END_VAR
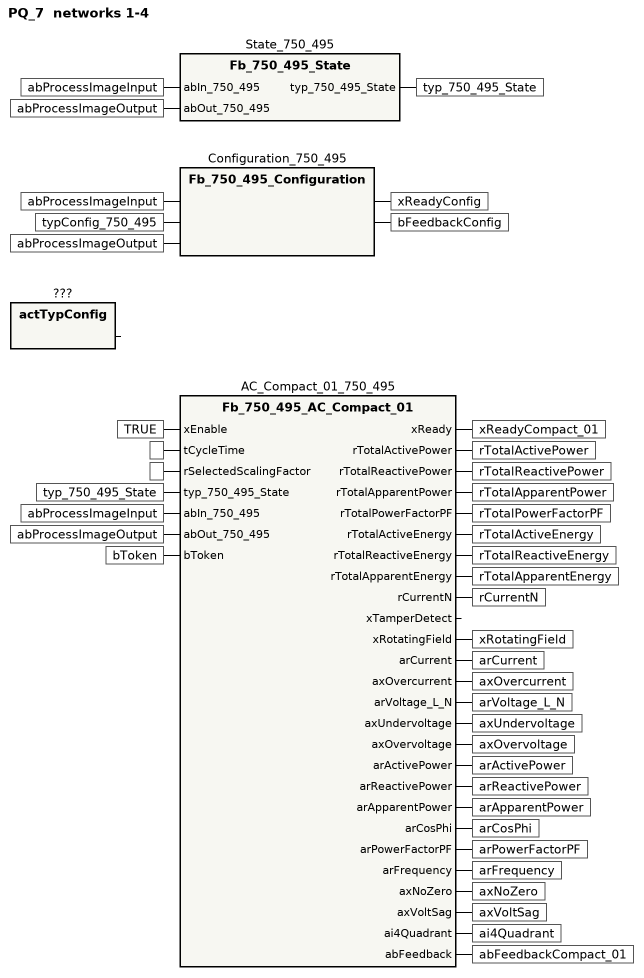
[picture p21: PQ_7 (FBD) networks 1-4]
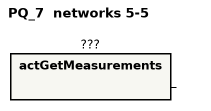
_FBD_ (* Function Block Diagram *)
NETWORK 1
	State_750_495:Fb_750_495_State(abIn_750_495: abProcessImageInput, abOut_750_495: abProcessImageOutput) => typ_750_495_State
NETWORK 2
	Configuration_750_495:Fb_750_495_Configuration(abProcessImageInput, typConfig_750_495, abProcessImageOutput, out 2 => bFeedbackConfig) => xReadyConfig
NETWORK 3
	???:actTypConfig()
NETWORK 4
	AC_Compact_01_750_495:Fb_750_495_AC_Compact_01(xEnable: TRUE, tCycleTime: , rSelectedScalingFactor: , typ_750_495_State: typ_750_495_State, abIn_750_495: abProcessImageInput, abOut_750_495: abProcessImageOutput, bToken: bToken, rTotalActivePower => rTotalActivePower, rTotalReactivePower => rTotalReactivePower, rTotalApparentPower => rTotalApparentPower, rTotalPowerFactorPF => rTotalPowerFactorPF, rTotalActiveEnergy => rTotalActiveEnergy, rTotalReactiveEnergy => rTotalReactiveEnergy, rTotalApparentEnergy => rTotalApparentEnergy, rCurrentN => rCurrentN, xRotatingField => xRotatingField, arCurrent => arCurrent, axOvercurrent => axOvercurrent, arVoltage_L_N => arVoltage_L_N, axUndervoltage => axUndervoltage, axOvervoltage => axOvervoltage, arActivePower => arActivePower, arReactivePower => arReactivePower, arApparentPower => arApparentPower, arCosPhi => arCosPhi, arPowerFactorPF => arPowerFactorPF, arFrequency => arFrequency, axNoZero => axNoZero, axVoltSag => axVoltSag, ai4Quadrant => ai4Quadrant, abFeedback => abFeedbackCompact_01) => xReadyCompact_01
NETWORK 5
	???:actGetMeasurements()
_END_FBD_
(* the same logic as Structured Text *)
(* Network 1 *)
State_750_495(abIn_750_495 := abProcessImageInput, abOut_750_495 := abProcessImageOutput);
typ_750_495_State := State_750_495.typ_750_495_State;
(* Network 2: see the listing above *)
(* Network 3: see the listing above *)
(* Network 4: see the listing above *)
(* Network 5: see the listing above *)
END_PROGRAM
ACTION actGetMeasurements:
arMeasurementsGroup7[1] := arActivePower[1];
arMeasurementsGroup7[2] := arActivePower[2];
arMeasurementsGroup7[3] := arActivePower[3];
arMeasurementsGroup7[4] := arReactivePower[1];
arMeasurementsGroup7[5] := arReactivePower[2];
arMeasurementsGroup7[6] := arReactivePower[3];
arMeasurementsGroup7[7] := arVoltage_L_N[1];
arMeasurementsGroup7[8] := arVoltage_L_N[2];
arMeasurementsGroup7[9] := arVoltage_L_N[3];
arMeasurementsGroup7[10] := arCurrent[1];
arMeasurementsGroup7[11] := arCurrent[2];
arMeasurementsGroup7[12] := arCurrent[3];
arMeasurementsGroup7[13] := arFrequency[1];
arMeasurementsGroup7[14] := arFrequency[2];
arMeasurementsGroup7[15] := arFrequency[3];
arMeasurementsGroup7[16] := rTotalActiveEnergy;
arMeasurementsGroup7[17] := BOOL_TO_REAL(xRotatingField);
arMeasurementsGroup7[18] := rTotalReactiveEnergy;
END_ACTION
ACTION actTypConfig:
typConfig_750_495.typChannelConfig[1].xEnableUserScaling:= TRUE;
typConfig_750_495.typChannelConfig[1].wCurrentTransformerRatio :=CurrentRatioPQ1;

typConfig_750_495.typChannelConfig[2].xEnableUserScaling:= TRUE;
typConfig_750_495.typChannelConfig[2].wCurrentTransformerRatio :=CurrentRatioPQ1;

typConfig_750_495.typChannelConfig[3].xEnableUserScaling:= TRUE;
typConfig_750_495.typChannelConfig[3].wCurrentTransformerRatio :=CurrentRatioPQ1;

typConfig_750_495.xWriteConfig := TRUE;
END_ACTION

(* POU 01. PowerQualityMeasurements/PQ_8, FBD *)
PROGRAM PQ_8
VAR
	abProcessImageInput	AT %IW96			: ARRAY[0..23] OF BYTE;
	abProcessImageOutput 	AT %QW104 		: ARRAY[0..23] OF BYTE;

	bToken										: BYTE;

	State_750_495 							: Fb_750_495_State;
		typ_750_495_State 						: typ_750_495_State;

	Configuration_750_495					: Fb_750_495_Configuration;
		typConfig_750_495						: typConfig_750_495;
		xReadyConfig								: BOOL;
		bFeedbackConfig							: BYTE;

	AC_Compact_01_750_495				: Fb_750_495_AC_Compact_01;
		rTotalActivePower							: REAL;
		rTotalReactivePower						: REAL;
		rTotalApparentPower						: REAL;
		rTotalPowerFactorPF						: REAL;
		rTotalActiveEnergy							: REAL;
		rTotalReactiveEnergy						: REAL;
		rTotalApparentEnergy						: REAL;
		rCurrentN									: REAL;
		xRotatingField								: BOOL;
		arCurrent									: ARRAY[1..3] OF REAL;
		axOvercurrent								: ARRAY[1..3] OF BOOL;
		arVoltage_L_N							: ARRAY[1..3] OF REAL;
		axUndervoltage							: ARRAY[1..3] OF BOOL;
		axOvervoltage								: ARRAY[1..3] OF BOOL;
		arActivePower								: ARRAY[1..3] OF REAL;
		arReactivePower							: ARRAY[1..3] OF REAL;
		arApparentPower							: ARRAY[1..3] OF REAL;
		arCosPhi									: ARRAY[1..3] OF REAL;
		arPowerFactorPF							: ARRAY[1..3] OF REAL;
		arFrequency								: ARRAY[1..3] OF REAL;
		axNoZero									: ARRAY[1..3] OF BOOL;
		axVoltSag									: ARRAY[1..3] OF BOOL;
		ai4Quadrant								: ARRAY[1..3] OF INT;

		xReadyCompact_01						: BOOL;
		abFeedbackCompact_01					: ARRAY[1..8] OF BYTE;


END_VAR
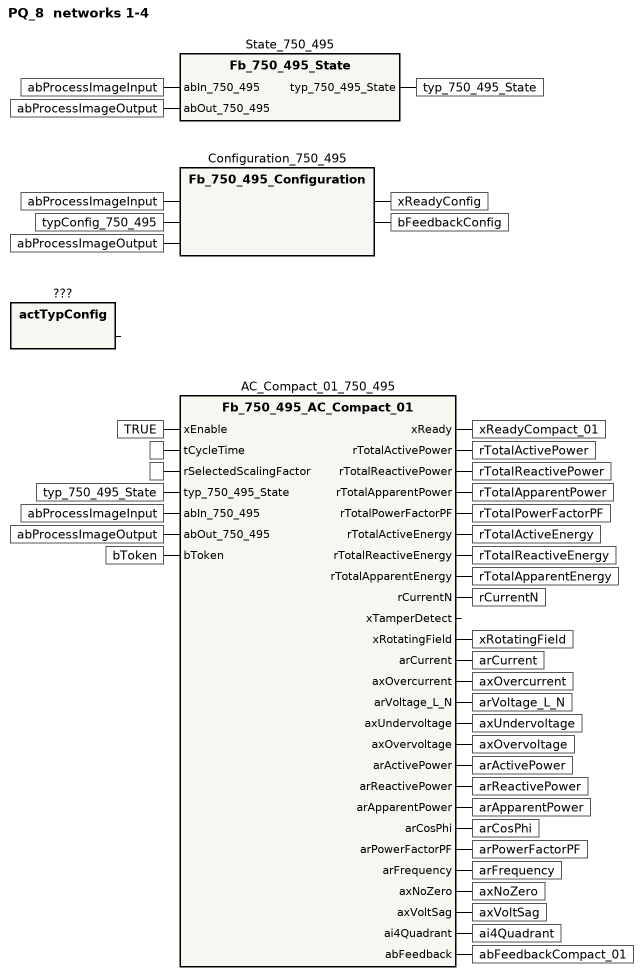
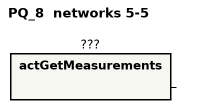
_FBD_ (* Function Block Diagram *)
NETWORK 1
	State_750_495:Fb_750_495_State(abIn_750_495: abProcessImageInput, abOut_750_495: abProcessImageOutput) => typ_750_495_State
NETWORK 2
	Configuration_750_495:Fb_750_495_Configuration(abProcessImageInput, typConfig_750_495, abProcessImageOutput, out 2 => bFeedbackConfig) => xReadyConfig
NETWORK 3
	???:actTypConfig()
NETWORK 4
	AC_Compact_01_750_495:Fb_750_495_AC_Compact_01(xEnable: TRUE, tCycleTime: , rSelectedScalingFactor: , typ_750_495_State: typ_750_495_State, abIn_750_495: abProcessImageInput, abOut_750_495: abProcessImageOutput, bToken: bToken, rTotalActivePower => rTotalActivePower, rTotalReactivePower => rTotalReactivePower, rTotalApparentPower => rTotalApparentPower, rTotalPowerFactorPF => rTotalPowerFactorPF, rTotalActiveEnergy => rTotalActiveEnergy, rTotalReactiveEnergy => rTotalReactiveEnergy, rTotalApparentEnergy => rTotalApparentEnergy, rCurrentN => rCurrentN, xRotatingField => xRotatingField, arCurrent => arCurrent, axOvercurrent => axOvercurrent, arVoltage_L_N => arVoltage_L_N, axUndervoltage => axUndervoltage, axOvervoltage => axOvervoltage, arActivePower => arActivePower, arReactivePower => arReactivePower, arApparentPower => arApparentPower, arCosPhi => arCosPhi, arPowerFactorPF => arPowerFactorPF, arFrequency => arFrequency, axNoZero => axNoZero, axVoltSag => axVoltSag, ai4Quadrant => ai4Quadrant, abFeedback => abFeedbackCompact_01) => xReadyCompact_01
NETWORK 5
	???:actGetMeasurements()
_END_FBD_
(* the same logic as Structured Text *)
(* Network 1 *)
State_750_495(abIn_750_495 := abProcessImageInput, abOut_750_495 := abProcessImageOutput);
typ_750_495_State := State_750_495.typ_750_495_State;
(* Network 2: see the listing above *)
(* Network 3: see the listing above *)
(* Network 4: see the listing above *)
(* Network 5: see the listing above *)
END_PROGRAM
ACTION actGetMeasurements:
arMeasurementsGroup8[1] := arActivePower[1];
arMeasurementsGroup8[2] := arActivePower[2];
arMeasurementsGroup8[3] := arActivePower[3];
arMeasurementsGroup8[4] := arReactivePower[1];
arMeasurementsGroup8[5] := arReactivePower[2];
arMeasurementsGroup8[6] := arReactivePower[3];
arMeasurementsGroup8[7] := arVoltage_L_N[1];
arMeasurementsGroup8[8] := arVoltage_L_N[2];
arMeasurementsGroup8[9] := arVoltage_L_N[3];
arMeasurementsGroup8[10] := arCurrent[1];
arMeasurementsGroup8[11] := arCurrent[2];
arMeasurementsGroup8[12] := arCurrent[3];
arMeasurementsGroup8[13] := arFrequency[1];
arMeasurementsGroup8[14] := arFrequency[2];
arMeasurementsGroup8[15] := arFrequency[3];
arMeasurementsGroup8[16] := rTotalActiveEnergy;
arMeasurementsGroup8[17] := BOOL_TO_REAL(xRotatingField);
arMeasurementsGroup8[18] := rTotalReactiveEnergy;
END_ACTION
ACTION actTypConfig:
typConfig_750_495.typChannelConfig[1].xEnableUserScaling:= TRUE;
typConfig_750_495.typChannelConfig[1].wCurrentTransformerRatio :=CurrentRatioPQ1;

typConfig_750_495.typChannelConfig[2].xEnableUserScaling:= TRUE;
typConfig_750_495.typChannelConfig[2].wCurrentTransformerRatio :=CurrentRatioPQ1;

typConfig_750_495.typChannelConfig[3].xEnableUserScaling:= TRUE;
typConfig_750_495.typChannelConfig[3].wCurrentTransformerRatio :=CurrentRatioPQ1;

typConfig_750_495.xWriteConfig := TRUE;
END_ACTION

(* POU 01. PowerQualityMeasurements/PQ_9, FBD *)
PROGRAM PQ_9
VAR
	abProcessImageInput	AT %IW108		: ARRAY[0..23] OF BYTE;
	abProcessImageOutput 	AT %QW116		: ARRAY[0..23] OF BYTE;

	bToken										: BYTE;

	State_750_495 							: Fb_750_495_State;
		typ_750_495_State 						: typ_750_495_State;

	Configuration_750_495					: Fb_750_495_Configuration;
		typConfig_750_495						: typConfig_750_495;
		xReadyConfig								: BOOL;
		bFeedbackConfig							: BYTE;

	AC_Compact_01_750_495				: Fb_750_495_AC_Compact_01;
		rTotalActivePower							: REAL;
		rTotalReactivePower						: REAL;
		rTotalApparentPower						: REAL;
		rTotalPowerFactorPF						: REAL;
		rTotalActiveEnergy							: REAL;
		rTotalReactiveEnergy						: REAL;
		rTotalApparentEnergy						: REAL;
		rCurrentN									: REAL;
		xRotatingField								: BOOL;
		arCurrent									: ARRAY[1..3] OF REAL;
		axOvercurrent								: ARRAY[1..3] OF BOOL;
		arVoltage_L_N							: ARRAY[1..3] OF REAL;
		axUndervoltage							: ARRAY[1..3] OF BOOL;
		axOvervoltage								: ARRAY[1..3] OF BOOL;
		arActivePower								: ARRAY[1..3] OF REAL;
		arReactivePower							: ARRAY[1..3] OF REAL;
		arApparentPower							: ARRAY[1..3] OF REAL;
		arCosPhi									: ARRAY[1..3] OF REAL;
		arPowerFactorPF							: ARRAY[1..3] OF REAL;
		arFrequency								: ARRAY[1..3] OF REAL;
		axNoZero									: ARRAY[1..3] OF BOOL;
		axVoltSag									: ARRAY[1..3] OF BOOL;
		ai4Quadrant								: ARRAY[1..3] OF INT;

		xReadyCompact_01						: BOOL;
		abFeedbackCompact_01					: ARRAY[1..8] OF BYTE;


END_VAR
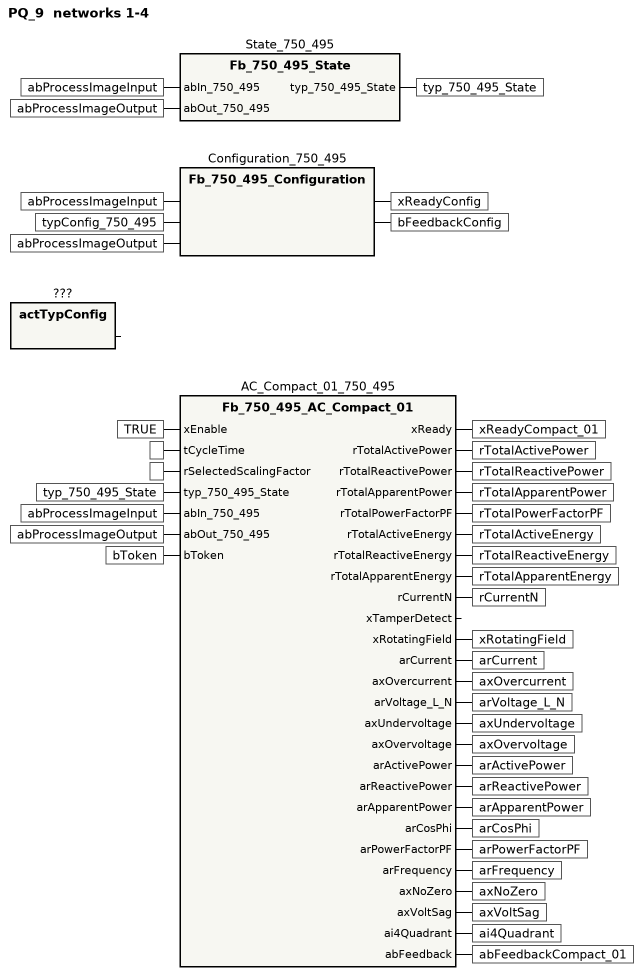
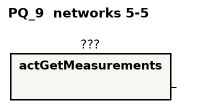
_FBD_ (* Function Block Diagram *)
NETWORK 1
	State_750_495:Fb_750_495_State(abIn_750_495: abProcessImageInput, abOut_750_495: abProcessImageOutput) => typ_750_495_State
NETWORK 2
	Configuration_750_495:Fb_750_495_Configuration(abProcessImageInput, typConfig_750_495, abProcessImageOutput, out 2 => bFeedbackConfig) => xReadyConfig
NETWORK 3
	???:actTypConfig()
NETWORK 4
	AC_Compact_01_750_495:Fb_750_495_AC_Compact_01(xEnable: TRUE, tCycleTime: , rSelectedScalingFactor: , typ_750_495_State: typ_750_495_State, abIn_750_495: abProcessImageInput, abOut_750_495: abProcessImageOutput, bToken: bToken, rTotalActivePower => rTotalActivePower, rTotalReactivePower => rTotalReactivePower, rTotalApparentPower => rTotalApparentPower, rTotalPowerFactorPF => rTotalPowerFactorPF, rTotalActiveEnergy => rTotalActiveEnergy, rTotalReactiveEnergy => rTotalReactiveEnergy, rTotalApparentEnergy => rTotalApparentEnergy, rCurrentN => rCurrentN, xRotatingField => xRotatingField, arCurrent => arCurrent, axOvercurrent => axOvercurrent, arVoltage_L_N => arVoltage_L_N, axUndervoltage => axUndervoltage, axOvervoltage => axOvervoltage, arActivePower => arActivePower, arReactivePower => arReactivePower, arApparentPower => arApparentPower, arCosPhi => arCosPhi, arPowerFactorPF => arPowerFactorPF, arFrequency => arFrequency, axNoZero => axNoZero, axVoltSag => axVoltSag, ai4Quadrant => ai4Quadrant, abFeedback => abFeedbackCompact_01) => xReadyCompact_01
NETWORK 5
	???:actGetMeasurements()
_END_FBD_
(* the same logic as Structured Text *)
(* Network 1 *)
State_750_495(abIn_750_495 := abProcessImageInput, abOut_750_495 := abProcessImageOutput);
typ_750_495_State := State_750_495.typ_750_495_State;
(* Network 2: see the listing above *)
(* Network 3: see the listing above *)
(* Network 4: see the listing above *)
(* Network 5: see the listing above *)
END_PROGRAM
ACTION actGetMeasurements:
arMeasurementsGroup9[1] := arActivePower[1];
arMeasurementsGroup9[2] := arActivePower[2];
arMeasurementsGroup9[3] := arActivePower[3];
arMeasurementsGroup9[4] := arReactivePower[1];
arMeasurementsGroup9[5] := arReactivePower[2];
arMeasurementsGroup9[6] := arReactivePower[3];
arMeasurementsGroup9[7] := arVoltage_L_N[1];
arMeasurementsGroup9[8] := arVoltage_L_N[2];
arMeasurementsGroup9[9] := arVoltage_L_N[3];
arMeasurementsGroup9[10] := arCurrent[1];
arMeasurementsGroup9[11] := arCurrent[2];
arMeasurementsGroup9[12] := arCurrent[3];
arMeasurementsGroup9[13] := arFrequency[1];
arMeasurementsGroup9[14] := arFrequency[2];
arMeasurementsGroup9[15] := arFrequency[3];
arMeasurementsGroup9[16] := rTotalActiveEnergy;
arMeasurementsGroup9[17] := BOOL_TO_REAL(xRotatingField);
arMeasurementsGroup9[18] := rTotalReactiveEnergy;
END_ACTION
ACTION actTypConfig:
typConfig_750_495.typChannelConfig[1].xEnableUserScaling:= TRUE;
typConfig_750_495.typChannelConfig[1].wCurrentTransformerRatio :=CurrentRatioPQ1;

typConfig_750_495.typChannelConfig[2].xEnableUserScaling:= TRUE;
typConfig_750_495.typChannelConfig[2].wCurrentTransformerRatio :=CurrentRatioPQ1;

typConfig_750_495.typChannelConfig[3].xEnableUserScaling:= TRUE;
typConfig_750_495.typChannelConfig[3].wCurrentTransformerRatio :=CurrentRatioPQ1;

typConfig_750_495.xWriteConfig := TRUE;
END_ACTION

(* POU 02. Batterybus Frequency to Analog Out/CHP_Controller, FBD *)
PROGRAM CHP_Controller
VAR
	RAMP_REAL: RAMP_REAL;
	Frequency_to_Analog_Out: Frequency_to_Analog_Out;
END_VAR
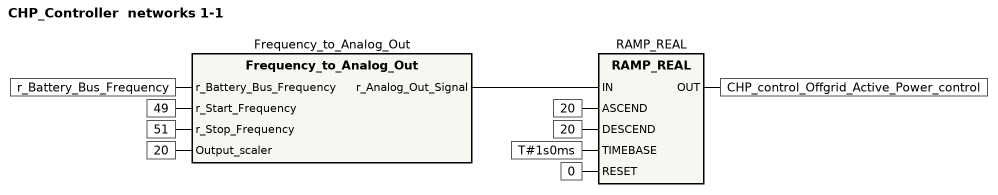
_FBD_ (* Function Block Diagram *)
NETWORK 1
	RAMP_REAL:RAMP_REAL(IN: Frequency_to_Analog_Out:Frequency_to_Analog_Out(r_Battery_Bus_Frequency: r_Battery_Bus_Frequency, r_Start_Frequency: 49, r_Stop_Frequency: 51, Output_scaler: 20), ASCEND: 20, DESCEND: 20, TIMEBASE: T#1s0ms, RESET: 0) => CHP_control_Offgrid_Active_Power_control
_END_FBD_
(* the same logic as Structured Text *)
(* Network 1 *)
Frequency_to_Analog_Out(r_Battery_Bus_Frequency := r_Battery_Bus_Frequency, r_Start_Frequency := 49, r_Stop_Frequency := 51, Output_scaler := 20);
RAMP_REAL(IN := Frequency_to_Analog_Out.r_Analog_Out_Signal, ASCEND := 20, DESCEND := 20, TIMEBASE := T#1s0ms, RESET := 0);
CHP_control_Offgrid_Active_Power_control := RAMP_REAL.OUT;
END_PROGRAM

(* POU 02. Batterybus Frequency to Analog Out/Frequency_to_Analog_Out, ST *)
FUNCTION_BLOCK Frequency_to_Analog_Out
VAR_INPUT
	r_Battery_Bus_Frequency						:	REAL;
	r_Start_Frequency								:	REAL:=49;
	r_Stop_Frequency								:	REAL:=51;
	Output_scaler										:	REAL:=1;
END_VAR

VAR_OUTPUT
	r_Analog_Out_Signal								:	REAL;
END_VAR

VAR

END_VAR
(* limit control range inbetween start/stop input*)
IF r_Start_Frequency < r_Stop_Frequency THEN
	IF r_Battery_Bus_Frequency < r_Start_Frequency THEN
			r_Battery_Bus_Frequency := r_Start_Frequency;
	END_IF
	IF r_Battery_Bus_Frequency > r_Stop_Frequency THEN
			r_Battery_Bus_Frequency := r_Stop_Frequency;
	END_IF
ELSE
	IF r_Battery_Bus_Frequency > r_Start_Frequency THEN
			r_Battery_Bus_Frequency := r_Start_Frequency;
	END_IF
	IF r_Battery_Bus_Frequency < r_Stop_Frequency THEN
			r_Battery_Bus_Frequency := r_Stop_Frequency;
	END_IF
END_IF

r_Analog_Out_Signal := (r_Battery_Bus_Frequency - r_Start_Frequency) / (r_Stop_Frequency - r_Start_Frequency) * Output_scaler;
END_FUNCTION_BLOCK

(* POU 02. Batterybus Frequency to Analog Out/EV_Controller, FBD *)
PROGRAM EV_Controller
VAR
	RAMP_REAL: RAMP_REAL;
	Frequency_to_Analog_Out: Frequency_to_Analog_Out;
END_VAR
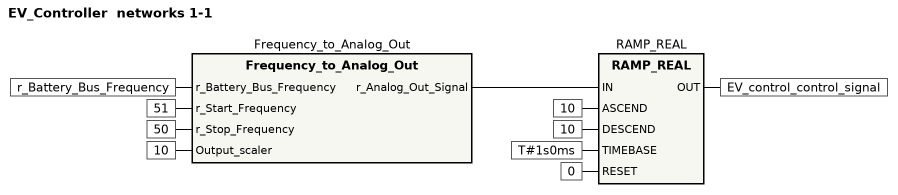
_FBD_ (* Function Block Diagram *)
NETWORK 1
	RAMP_REAL:RAMP_REAL(IN: Frequency_to_Analog_Out:Frequency_to_Analog_Out(r_Battery_Bus_Frequency: r_Battery_Bus_Frequency, r_Start_Frequency: 51, r_Stop_Frequency: 50, Output_scaler: 10), ASCEND: 10, DESCEND: 10, TIMEBASE: T#1s0ms, RESET: 0) => EV_control_control_signal
_END_FBD_
(* the same logic as Structured Text *)
(* Network 1 *)
Frequency_to_Analog_Out(r_Battery_Bus_Frequency := r_Battery_Bus_Frequency, r_Start_Frequency := 51, r_Stop_Frequency := 50, Output_scaler := 10);
RAMP_REAL(IN := Frequency_to_Analog_Out.r_Analog_Out_Signal, ASCEND := 10, DESCEND := 10, TIMEBASE := T#1s0ms, RESET := 0);
EV_control_control_signal := RAMP_REAL.OUT;
END_PROGRAM

(* POU 02. Batterybus Frequency to Analog Out/Mixer_Controller, FBD *)
PROGRAM Mixer_Controller
VAR
	RAMP_REAL: RAMP_REAL;
	Frequency_to_Analog_Out: Frequency_to_Analog_Out;
END_VAR
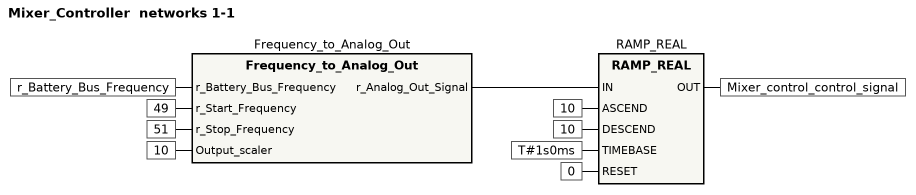
_FBD_ (* Function Block Diagram *)
NETWORK 1
	RAMP_REAL:RAMP_REAL(IN: Frequency_to_Analog_Out:Frequency_to_Analog_Out(r_Battery_Bus_Frequency: r_Battery_Bus_Frequency, r_Start_Frequency: 49, r_Stop_Frequency: 51, Output_scaler: 10), ASCEND: 10, DESCEND: 10, TIMEBASE: T#1s0ms, RESET: 0) => Mixer_control_control_signal
_END_FBD_
(* the same logic as Structured Text *)
(* Network 1 *)
Frequency_to_Analog_Out(r_Battery_Bus_Frequency := r_Battery_Bus_Frequency, r_Start_Frequency := 49, r_Stop_Frequency := 51, Output_scaler := 10);
RAMP_REAL(IN := Frequency_to_Analog_Out.r_Analog_Out_Signal, ASCEND := 10, DESCEND := 10, TIMEBASE := T#1s0ms, RESET := 0);
Mixer_control_control_signal := RAMP_REAL.OUT;
END_PROGRAM

(* POU PLC_PRG, FBD *)
PROGRAM PLC_PRG
(*
  Function: 	Reading a CSV file
  Description: 	This project shows a functionblock which reads data from a CSV file into an array.
				Each line in the CSV contains a description and a real value.
				Each parameter  is terminated by CR LF.

---- Example CSV File -----

A_Value;245345
B_Value;0							
C_Value;8.3							
D_Value;-123439.3 						
E_Value;1						*)

VAR
	xLoad					: 	BOOL; (* Initiate load operation *)
	xSave					: 	BOOL; (* Initiate save operation *)
	sLoadStatus			: 	STRING; (* Feedback on load *)
	sSaveStatus			: 	STRING; (* Feedback on save *)
	ConfigData			: 	ARRAY [1..iMaxParams] OF  typCSV; (* Structure with the config data being loaded or saved *)
	sFileName			: 	STRING := 'config.csv'; (* Working Filename *)
	bSeperator 			: 	BYTE := 59; (* Semicolon (;) is the seperator between parameter and value. *)
	iError					: 	INT; (* Error Code for Save *)
	xWriteToSD			: 	BOOL := TRUE; (* User selectable location for file operation, on = 750-880 SD, off = internal flash *)
	sFilePath				: 	STRING; (* SD card is S:\, Internal Path is blank, but this points to the PLC folder *)
	sFilePath_Name		: 	STRING; (* Complete path + filename *)

	xReadFirstCycle		:	BOOL := TRUE;

	SetIPConfig				:	configToolFB;
	SetIP						:	configToolFB;
	SetSubnet					:	configToolFB;
	SetGateway				:	configToolFB;
	SetNTP					:	configToolFB;
	SetNTPEnable			:	configToolFB;
	SetSNMPName			:	configToolFB;
	SetSNMPDescription		:	configToolFB;
	SetSNMPLocation			:	configToolFB;
	SetSNMPContact			:	configToolFB;

	GetIPConfig				:	configToolFB;
	GetIP						:	configToolFB;
	GetSubnet					:	configToolFB;
	GetGateway				:	configToolFB;
	GetNTP					:	configToolFB;
	GetSNMPName			:	configToolFB;
	GetSNMPDescription		:	configToolFB;
	GetSNMPLocation		:	configToolFB;
	GetSNMPContact			:	configToolFB;
	GetFirmware				:	configToolFB;
	GetMACAddress			:	configToolFB;
	GetProjectDate			:	configToolFB;
	GetProjectDescription	:	configToolFB;
	GetProjectVersion			:	configToolFB;

	stSetIPConfigCallstring				:	STRING(80);
	stSetIPCallstring						:	STRING(80);
	stSetSubnetCallstring				:	STRING(80);
	stSetGatewayCallstring				:	STRING(80);
	stSetNTPCallstring					:	STRING(80);

	iSetIPConfigCallstringResult			:	INT;
	iSetIPCallstringResult				:	INT;
	iSetSubnetCallstringResult			:	INT;
	iSetGatewayCallstringResult			:	INT;
	iSetNTPCallstringResult				: 	INT;
	iSetNTPEnabledCallstringResult	:	INT;

	iGetIPConfigCallstringResult			:	INT;
	iGetIPCallstringResult				:	INT;
	iGetSubnetCallstringResult			:	INT;
	iGetGatewayCallstringResult			:	INT;
	iGetNTPCallstringResult				: 	INT;
	iGetNTPEnabledCallstringResult	:	INT;

	iGetFirmwareCallstringResult				:	INT;
	iGetMACAddressCallstringResult			:	INT;
	iGetProjectDateCallstringResult				:	INT;
	iGetProjectDescriptionCallstringResult		:	INT;
	iGetProjectVersionCallstringResult			:	INT;

	stGetIPConfigCallstring				:	STRING(80);
	stGetIPCallstring						:	STRING(80);
	stGetSubnetCallstring				:	STRING(80);
	stGetGatewayCallstring				:	STRING(80);
	stGetNTPCallstring					:	STRING(80);

	stSetIPConfigResult					:	STRING(80);
	stSetIPResult							:	STRING(80);
	stSetSubnetResult					:	STRING(80);
	stSetGatewayResult					:	STRING(80);
	stSetNTPResult						:	STRING(80);

	stGetIPConfigResult					:	STRING(80);
	stGetIPResult							:	STRING(80);
	stGetSubnetResult					:	STRING(80);
	stGetGatewayResult					:	STRING(80);
	stGetNTPResult						:	STRING(80);

	stSetSNMPNameDeviceCallstring					:	STRING(80);
	stSetSNMPDescriptionCallstring						:	STRING(80);
	stSetSNMPPhysicalLocationCallstring				:	STRING(80);
	stSetSNMPContactCallstring							:	STRING(80);

	stGetSNMPNameDeviceResult						:	STRING(80);
	stGetSNMPDescriptionResult						:	STRING(80);
	stGetSNMPPhysicalLocationResult					:	STRING(80);
	stGetSNMPContactResult							:	STRING(80);

	stGetFirmwareResult									:	STRING(80);
	stGetMACAddressResult								:	STRING(80);
	stGetProjectDateResult								:	STRING(80);
	stGetProjectDescriptionResult						:	STRING(80);
	stGetProjectVersionResult							:	STRING(80);

	iSetSNMPNameDeviceCallstringResult				:	INT;
	iSetSNMPDescriptionCallstringResult				:	INT;
	iSetSNMPPhysicalLocationCallstringResult			:	INT;
	iSetSNMPContactCallstringResult					:	INT;

	iGetSNMPNameDeviceCallstringResult				:	INT;
	iGetSNMPDescriptionCallstringResult				:	INT;
	iGetSNMPPhysicalLocationCallstringResult			:	INT;
	iGetSNMPContactCallstringResult					:	INT;

	CurrentTimeDate										:	STRING;

END_VAR
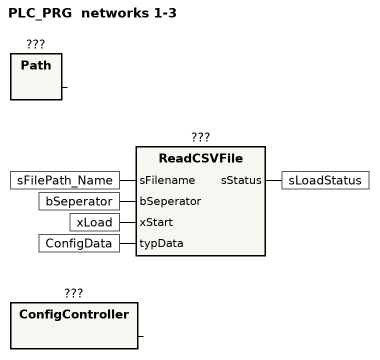
_FBD_ (* Function Block Diagram *)
NETWORK 1
	???:Path()
NETWORK 2
	???:ReadCSVFile(sFilename: sFilePath_Name, bSeperator: bSeperator, xStart: xLoad, typData: ConfigData) => sLoadStatus
NETWORK 3
	???:ConfigController()
_END_FBD_
END_PROGRAM
ACTION ConfigController:
IF xReadFirstCycle = TRUE THEN

	(*xLoad := TRUE;*)

	IF sLoadStatus = 'Data read OK' THEN
	
		(* Set Ethernet settings of controller *)
		
		(* Set static IP-Address*)
		
		
			SetIPConfig(
			bEnable:= TRUE,
			stCallString:= 'config_interfaces interface=X1 config-type=static state=enabled',
			stResultString=> stSetIPConfigResult,
			iFbResult=> iSetIPCallstringResult );
		
		(* Set IP-Address of controller *)
		
			stSetIPCallstring := CONCAT('config_interfaces interface X1 ip-address=',stIPAddressEthernet);
		
			SetIP(
			bEnable:= TRUE,
			stCallString:= stSetIPCallstring ,
			stResultString=> stSetIPResult,
			iFbResult=> iSetIPCallstringResult );
		
		(* Set Subnet-Address of controller *)
		
			stSetSubnetCallstring := CONCAT('config_interfaces interface X1 subnet-mask=',stIPAddressSubnet);
		
			SetSubnet(
			bEnable:= TRUE,
			stCallString:= stSetSubnetCallstring ,
			iFbResult=> iSetSubnetCallstringResult );
		
		(* Set Gateway-Address of controller *)
		
			stSetGatewayCallstring := CONCAT('config_default_gateway interface=X1 default-gateway-value=', stIPAddressGateway);
		
			SetGateway(
			bEnable:= TRUE,
			stCallString:= stSetGatewayCallstring ,
			iFbResult=> iSetGatewayCallstringResult );
		
		(* Set NTP-Address of controller *)
		
			SetNTPEnable(
			bEnable:= TRUE,
			stCallString:= 'config_sntp state=enabled' ,
			iFbResult=> iSetNTPEnabledCallstringResult );
		
			stSetNTPCallstring := CONCAT('config_sntp time-server=',stIPAddressNTP);
		
			SetNTP(
			bEnable:= TRUE,
			stCallString:= stSetNTPCallstring ,
			iFbResult=> iSetNTPCallstringResult );
		
		(* Set SNMP-configuration of the controller *)
		
		(* Set SNMP-description of the controller *)
		
			stSetSNMPDescriptionCallstring := CONCAT('config_snmp description=',stSNMPDescription);
		
			SetSNMPDescription(
			bEnable:= TRUE,
			stCallString:= stSetSNMPDescriptionCallstring,
			iFbResult=> iSetSNMPDescriptionCallstringResult );
		
		(* Set SNMP-name of the controller *)
		
			stSetSNMPNameDeviceCallstring := CONCAT('config_snmp device-name=',stSNMPNameDevice);
		
			SetSNMPName(
			bEnable:= TRUE,
			stCallString:= stSetSNMPNameDeviceCallstring,
			iFbResult=> iSetSNMPNameDeviceCallstringResult );
		
		(* Set SNMP-location of the controller *)

			stSetSNMPPhysicalLocationCallstring := CONCAT('config_snmp physical-location=',stSNMPPhysicalLocation);
		
			SetSNMPLocation(
			bEnable:= TRUE,
			stCallString:= stSetSNMPPhysicalLocationCallstring,
			iFbResult=> iSetSNMPPhysicalLocationCallstringResult);
		
		(* Set SNMP-contact information of the controller *)
		
			stSetSNMPContactCallstring := CONCAT('config_snmp contact=',stSNMPcontact);
		
			SetSNMPContact(
			bEnable:= TRUE,
			stCallString:= stSetSNMPContactCallstring,
			iFbResult=> iSetSNMPContactCallstringResult);
		
			xReadFirstCycle := FALSE;
			xLoad := FALSE;

	END_IF

END_IF

(* Get Ethernet settings of controller *)

(* Get IP-configuration of controller *)

	GetIPConfig(
	bEnable:= TRUE,
	stCallString:= 'get_eth_config X1 config-type' ,
	stResultString=> stGetIPConfigResult,
	iFbResult=> iGetIPConfigCallstringResult );

(* Get IP-Address of controller *)

	GetIP(
	bEnable:= TRUE,
	stCallString:= 'get_eth_config X1 ip-address' ,
	stResultString=> stGetIPResult,
	iFbResult=> iGetIPCallstringResult );

(* Get Subnet-Address of controller *)

	GetSubnet(
	bEnable:= TRUE,
	stCallString:= 'get_eth_config X1 subnet-mask' ,
	stResultString=> stGetSubnetResult,
	iFbResult=> iGetSubnetCallstringResult );

(* Get Gateway-Address of controller *)

	GetGateway(
	bEnable:= TRUE,
	stCallString:= 'get_eth_config X1 default-gateway' ,
	stResultString=> stGetGatewayResult,
	iFbResult=> iGetGatewayCallstringResult );

(* Get NTP-Address of controller *)

	GetNTP(
	bEnable:= TRUE,
	stCallString:= 'get_ntp_config time-server' ,
	stResultString=> stGetNTPResult,
	iFbResult=> iGetNTPCallstringResult );

(* Get SNMP-configuration of the controller *)

(* Get SNMP-description of the controller *)

	GetSNMPDescription(
	bEnable:= TRUE,
	stCallString:= 'get_snmp_data description',
	stResultString=> stGetSNMPDescriptionResult,
	iFbResult=> iGetSNMPDescriptionCallstringResult );

(* Get SNMP-description of the controller *)

	GetSNMPName(
	bEnable:= TRUE,
	stCallString:= 'get_snmp_data device-name',
	stResultString=> stGetSNMPNameDeviceResult,
	iFbResult=> iGetSNMPNameDeviceCallstringResult );

(* Get SNMP-location of the controller *)

	GetSNMPLocation(
	bEnable:= TRUE,
	stCallString:= 'get_snmp_data physical-location',
	stResultString=> stGetSNMPPhysicalLocationResult,
	iFbResult=> iGetSNMPPhysicalLocationCallstringResult);

(* Get SNMP-contact information of the controller *)

	GetSNMPContact(
	bEnable:= TRUE,
	stCallString:= 'get_snmp_data contact',
	stResultString=> stGetSNMPContactResult,
	iFbResult=> iGetSNMPContactCallstringResult);

(* Get Firmware information of the controller *)

	GetFirmware(
	bEnable:= TRUE,
	stCallString:= 'get_coupler_details firmware-revision',
	stResultString=> stGetFirmwareResult,
	iFbResult=> iGetFirmwareCallstringResult);

(* Get MAC-Address of the controller *)

	GetMACAddress(
	bEnable:= TRUE,
	stCallString:= 'get_actual_eth_config X1 mac-address',
	stResultString=> stGetMACAddressResult,
	iFbResult=> iGetMACAddressCallstringResult);

(* Get Project Date of the controller *)

	GetProjectDate(
	bEnable:= TRUE,
	stCallString:= 'get_rts_info project date',
	stResultString=> stGetProjectDateResult,
	iFbResult=> iGetProjectDateCallstringResult);

(* Get Project Description of the controller *)

	GetProjectDescription(
	bEnable:= TRUE,
	stCallString:= 'get_rts_info project description',
	stResultString=> stGetProjectDescriptionResult,
	iFbResult=> iGetProjectDescriptionCallstringResult);

(* Get Project version of the controller *)

	GetProjectVersion(
	bEnable:= TRUE,
	stCallString:= 'get_rts_info project version',
	stResultString=> stGetProjectVersionResult,
	iFbResult=> iGetProjectVersionCallstringResult);

	CurrentTimeDate := Date_Time();
END_ACTION
ACTION Path:
IF xWriteToSD THEN
	sFilePath := '/media/sd/';
ELSE
	sFilePath := '';
END_IF
sFilePath_Name := CONCAT(sFilePath, sFileName);
END_ACTION
ACTION SetParam:
	stIPAddressEthernet := ConfigData[1].Parameter[1];
	stIPAddressSubnet  := ConfigData[2].Parameter[1];
	stIPAddressGateway  := ConfigData[3].Parameter[1];
	stIPAddressNTP := ConfigData[4].Parameter[1];

	stSNMPNameDevice := ConfigData[5].Parameter[1];
	stSNMPDescription := ConfigData[6].Parameter[1];
	stSNMPPhysicalLocation := ConfigData[7].Parameter[1];
	stSNMPContact := ConfigData[8].Parameter[1];
END_ACTION

(* POU 08. SD CARD logging/ReadCSVFile, ST *)
PROGRAM ReadCSVFile
VAR_INPUT
	sFilename		:STRING;
	bSeperator		:BYTE:=59;(*seperator semicolon:59=;*)
END_VAR
VAR_IN_OUT
	xStart			:BOOL;
	typData			:ARRAY [1..iMaxParams] OF  typCSV;
END_VAR
VAR_OUTPUT
	sStatus			:STRING;
END_VAR
VAR
	bEndOfFile		:BYTE:=13;
	FileIdent		:DWORD;
	rawdata			:ARRAY[0..gc_RawDataSize] OF BYTE;
	filesizev		:DINT;
	tempstring		:STRING;
	startposition	:INT;
	i				:INT;
	j				:INT;
	k				:INT;
END_VAR
IF xStart THEN
	FileIdent:=SysFileOpen(FileName:=sFilename, Mode:='r');
	IF fileident<>0 THEN
		SysFileRead(File:=Fileident, Buffer:=ADR(rawdata), Size:=SIZEOF(rawdata));
		filesizev:=SysFileGetSize(FileName:=sFilename);
		IF filesizev>gc_RawDataSize THEN
			filesizev:=gc_RawDataSize;
		END_IF
		SysFileClose(File:=fileident);(*this function is blocking*)
	ELSE
		sStatus:='File does not exist';
		xStart:=FALSE;
		RETURN;(*no such file available*)
	END_IF
(*copy data to typData array*)
	startposition:=0;
	i:=0;
	FOR j:=1 TO iMaxParams DO
		(*First value in dataset is of type DT. The following value is seperated by bSeperator*)
		WHILE rawdata[startposition+i]<>bSeperator DO
			i:=i+1;
		END_WHILE
		rawdata[startposition+i]:=0;
		MEMCPY(pSourceAddress:=ADR(rawdata[startposition]), pDestinationAddress:=ADR(tempstring), BytesToCopy:=i+1);
		typdata[j].sDescription:=tempstring;
		startposition:=startposition+i+1;
		i:=0;
		(*The parameter values are of type word. The following values are seperated by bSeperator*)
		FOR k:=1 TO gc_ParameterCount-1 DO
			WHILE rawdata[startposition+i]<>bSeperator DO
				i:=i+1;
			END_WHILE
			rawdata[startposition+i]:=0;
			MEMCPY(pSourceAddress:=ADR(rawdata[startposition]), pDestinationAddress:=ADR(tempstring), BytesToCopy:=i+1);
			typdata[j].Parameter[k]:=(tempstring);
			startposition:=startposition+i+1;
			i:=0;
		END_FOR
		(*Copying the last parameter from typ word. The data set is terminated by CR LF*)
		WHILE rawdata[startposition+i]<>bEndOfFile DO
			i:=i+1;
		END_WHILE
		rawdata[startposition+i]:=0;
		MEMCPY(pSourceAddress:=ADR(rawdata[startposition]), pDestinationAddress:=ADR(tempstring), BytesToCopy:=i+1);
		typdata[j].Parameter[k]:=(tempstring);
		startposition:=startposition+i+2;(*The data set is terminated by CR LF(13,10)*)
		i:=0;
	END_FOR
(*copy data to typData array finished*)
	sStatus:='Data read OK';
	xStart:=FALSE;
END_IF
END_PROGRAM

(* POU 07. Signal Lights/error_lights, ST *)
PROGRAM error_lights
VAR
END_VAR
	Control_panel_status_operational_led := 1;
	Control_panel_status_warning_led	:=0;
	Control_panel_status_error_led := 0;

IF arMeasurementsGroupA[6] < 220 THEN
		Control_panel_status_warning_led := 1;  (* Low Grid Voltage *)
END_IF


(*--------------------------------------------------------------------------------------------------------------------------------------------------*)
IF Group1_3F_Auto_relay_control_battery_bus <> Group1_3F_relay_state_battery_bus  THEN
		Control_panel_status_error_led := 1;
END_IF


IF Group1_3F_Auto_relay_control_grid_bus <> Group1_3F_relay_state_grid_bus  THEN
		Control_panel_status_error_led := 1;
END_IF



(*--------------------------------------------------------------------------------------------------------------------------------------------------*)
IF Group2_3F_Auto_relay_control_battery_bus <> Group2_3F_relay_state_battery_bus  THEN
		Control_panel_status_error_led := 1;
END_IF


IF Group2_3F_Auto_relay_control_grid_bus <> Group2_3F_relay_state_grid_bus  THEN
		Control_panel_status_error_led := 1;
END_IF


(*--------------------------------------------------------------------------------------------------------------------------------------------------*)
IF Group3_3F_Auto_relay_control_battery_bus <> Group3_3F_relay_state_battery_bus  THEN
		Control_panel_status_error_led := 1;
END_IF


IF Group3_3F_Auto_relay_control_grid_bus <> Group3_3F_relay_state_grid_bus  THEN
		Control_panel_status_error_led := 1;
END_IF


(*--------------------------------------------------------------------------------------------------------------------------------------------------*)
IF Group4_3F_Auto_relay_control_battery_bus <> Group4_3F_relay_state_battery_bus  THEN
		Control_panel_status_error_led := 1;
END_IF


IF Group4_3F_Auto_relay_control_grid_bus <> Group4_3F_relay_state_grid_bus  THEN
		Control_panel_status_error_led := 1;
END_IF


(*--------------------------------------------------------------------------------------------------------------------------------------------------*)
IF Group5_3F_Auto_relay_control_battery_bus <> Group5_3F_relay_state_battery_bus  THEN
		Control_panel_status_error_led := 1;
END_IF


IF Group5_3F_Auto_relay_control_grid_bus <> Group5_3F_relay_state_grid_bus  THEN
		Control_panel_status_error_led := 1;
END_IF


(*--------------------------------------------------------------------------------------------------------------------------------------------------*)
IF Group6_3F_Auto_relay_control_battery_bus <> Group6_3F_relay_state_battery_bus  THEN
		Control_panel_status_error_led := 1;
END_IF


IF Group6_3F_Auto_relay_control_grid_bus <> Group6_3F_relay_state_grid_bus  THEN
		Control_panel_status_error_led := 1;
END_IF


(*--------------------------------------------------------------------------------------------------------------------------------------------------*)
IF Group7_3F_Auto_relay_control_battery_bus <> Group7_3F_relay_state_battery_bus  THEN
		Control_panel_status_error_led := 1;
END_IF


IF Group7_3F_Auto_relay_control_grid_bus <> Group7_3F_relay_state_grid_bus  THEN
		Control_panel_status_error_led := 1;
END_IF


(*--------------------------------------------------------------------------------------------------------------------------------------------------*)
IF Group8_3F_Auto_relay_control_battery_bus <> Group8_3F_relay_state_battery_bus  THEN
		Control_panel_status_error_led := 1;
END_IF


IF Group8_3F_Auto_relay_control_grid_bus <> Group8_3F_relay_state_grid_bus  THEN
		Control_panel_status_error_led := 1;
END_IF


(*--------------------------------------------------------------------------------------------------------------------------------------------------*)
IF Group9_3F_Auto_relay_control_battery_bus <> Group9_3F_relay_state_battery_bus  THEN
		Control_panel_status_error_led := 1;
END_IF


IF Group9_3F_Auto_relay_control_grid_bus <> Group9_3F_relay_state_grid_bus  THEN
		Control_panel_status_error_led := 1;
END_IF
END_PROGRAM

(* POU 04. Frequency based Bus Select/Group3, FBD *)
PROGRAM Group3
VAR
	Switch3:fbSwitchRelaysBatOrGridBus;
END_VAR
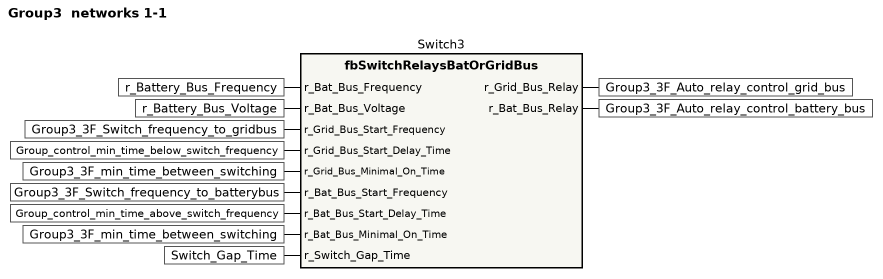
_FBD_ (* Function Block Diagram *)
NETWORK 1
	Switch3:fbSwitchRelaysBatOrGridBus(r_Bat_Bus_Frequency: r_Battery_Bus_Frequency, r_Bat_Bus_Voltage: r_Battery_Bus_Voltage, r_Grid_Bus_Start_Frequency: Group3_3F_Switch_frequency_to_gridbus, r_Grid_Bus_Start_Delay_Time: Group_control_min_time_below_switch_frequency, r_Grid_Bus_Minimal_On_Time: Group3_3F_min_time_between_switching, r_Bat_Bus_Start_Frequency: Group3_3F_Switch_frequency_to_batterybus, r_Bat_Bus_Start_Delay_Time: Group_control_min_time_above_switch_frequency, r_Bat_Bus_Minimal_On_Time: Group3_3F_min_time_between_switching, r_Switch_Gap_Time: Switch_Gap_Time, r_Bat_Bus_Relay => Group3_3F_Auto_relay_control_battery_bus) => Group3_3F_Auto_relay_control_grid_bus
_END_FBD_
(* the same logic as Structured Text *)
(* Network 1 *)
Switch3(r_Bat_Bus_Frequency := r_Battery_Bus_Frequency, r_Bat_Bus_Voltage := r_Battery_Bus_Voltage, r_Grid_Bus_Start_Frequency := Group3_3F_Switch_frequency_to_gridbus, r_Grid_Bus_Start_Delay_Time := Group_control_min_time_below_switch_frequency, r_Grid_Bus_Minimal_On_Time := Group3_3F_min_time_between_switching, r_Bat_Bus_Start_Frequency := Group3_3F_Switch_frequency_to_batterybus, r_Bat_Bus_Start_Delay_Time := Group_control_min_time_above_switch_frequency, r_Bat_Bus_Minimal_On_Time := Group3_3F_min_time_between_switching, r_Switch_Gap_Time := Switch_Gap_Time);
Group3_3F_Auto_relay_control_battery_bus := Switch3.r_Bat_Bus_Relay;
Group3_3F_Auto_relay_control_grid_bus := Switch3.r_Grid_Bus_Relay;
END_PROGRAM

(* POU 04. Frequency based Bus Select/Group4, FBD *)
PROGRAM Group4
VAR
	Switch4:fbSwitchRelaysBatOrGridBus;
END_VAR
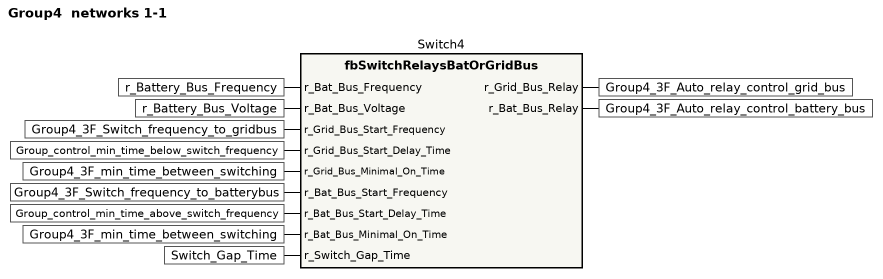
_FBD_ (* Function Block Diagram *)
NETWORK 1
	Switch4:fbSwitchRelaysBatOrGridBus(r_Bat_Bus_Frequency: r_Battery_Bus_Frequency, r_Bat_Bus_Voltage: r_Battery_Bus_Voltage, r_Grid_Bus_Start_Frequency: Group4_3F_Switch_frequency_to_gridbus, r_Grid_Bus_Start_Delay_Time: Group_control_min_time_below_switch_frequency, r_Grid_Bus_Minimal_On_Time: Group4_3F_min_time_between_switching, r_Bat_Bus_Start_Frequency: Group4_3F_Switch_frequency_to_batterybus, r_Bat_Bus_Start_Delay_Time: Group_control_min_time_above_switch_frequency, r_Bat_Bus_Minimal_On_Time: Group4_3F_min_time_between_switching, r_Switch_Gap_Time: Switch_Gap_Time, r_Bat_Bus_Relay => Group4_3F_Auto_relay_control_battery_bus) => Group4_3F_Auto_relay_control_grid_bus
_END_FBD_
(* the same logic as Structured Text *)
(* Network 1 *)
Switch4(r_Bat_Bus_Frequency := r_Battery_Bus_Frequency, r_Bat_Bus_Voltage := r_Battery_Bus_Voltage, r_Grid_Bus_Start_Frequency := Group4_3F_Switch_frequency_to_gridbus, r_Grid_Bus_Start_Delay_Time := Group_control_min_time_below_switch_frequency, r_Grid_Bus_Minimal_On_Time := Group4_3F_min_time_between_switching, r_Bat_Bus_Start_Frequency := Group4_3F_Switch_frequency_to_batterybus, r_Bat_Bus_Start_Delay_Time := Group_control_min_time_above_switch_frequency, r_Bat_Bus_Minimal_On_Time := Group4_3F_min_time_between_switching, r_Switch_Gap_Time := Switch_Gap_Time);
Group4_3F_Auto_relay_control_battery_bus := Switch4.r_Bat_Bus_Relay;
Group4_3F_Auto_relay_control_grid_bus := Switch4.r_Grid_Bus_Relay;
END_PROGRAM

(* POU 04. Frequency based Bus Select/Group5, FBD *)
PROGRAM Group5
VAR
	Switch5:fbSwitchRelaysBatOrGridBus;
END_VAR
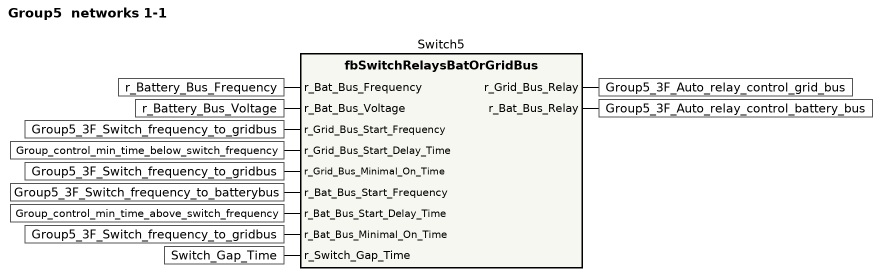
_FBD_ (* Function Block Diagram *)
NETWORK 1
	Switch5:fbSwitchRelaysBatOrGridBus(r_Bat_Bus_Frequency: r_Battery_Bus_Frequency, r_Bat_Bus_Voltage: r_Battery_Bus_Voltage, r_Grid_Bus_Start_Frequency: Group5_3F_Switch_frequency_to_gridbus, r_Grid_Bus_Start_Delay_Time: Group_control_min_time_below_switch_frequency, r_Grid_Bus_Minimal_On_Time: Group5_3F_Switch_frequency_to_gridbus, r_Bat_Bus_Start_Frequency: Group5_3F_Switch_frequency_to_batterybus, r_Bat_Bus_Start_Delay_Time: Group_control_min_time_above_switch_frequency, r_Bat_Bus_Minimal_On_Time: Group5_3F_Switch_frequency_to_gridbus, r_Switch_Gap_Time: Switch_Gap_Time, r_Bat_Bus_Relay => Group5_3F_Auto_relay_control_battery_bus) => Group5_3F_Auto_relay_control_grid_bus
_END_FBD_
(* the same logic as Structured Text *)
(* Network 1 *)
Switch5(r_Bat_Bus_Frequency := r_Battery_Bus_Frequency, r_Bat_Bus_Voltage := r_Battery_Bus_Voltage, r_Grid_Bus_Start_Frequency := Group5_3F_Switch_frequency_to_gridbus, r_Grid_Bus_Start_Delay_Time := Group_control_min_time_below_switch_frequency, r_Grid_Bus_Minimal_On_Time := Group5_3F_Switch_frequency_to_gridbus, r_Bat_Bus_Start_Frequency := Group5_3F_Switch_frequency_to_batterybus, r_Bat_Bus_Start_Delay_Time := Group_control_min_time_above_switch_frequency, r_Bat_Bus_Minimal_On_Time := Group5_3F_Switch_frequency_to_gridbus, r_Switch_Gap_Time := Switch_Gap_Time);
Group5_3F_Auto_relay_control_battery_bus := Switch5.r_Bat_Bus_Relay;
Group5_3F_Auto_relay_control_grid_bus := Switch5.r_Grid_Bus_Relay;
END_PROGRAM

(* POU 04. Frequency based Bus Select/Group6, FBD *)
PROGRAM Group6
VAR
	Switch6:fbSwitchRelaysBatOrGridBus;
END_VAR
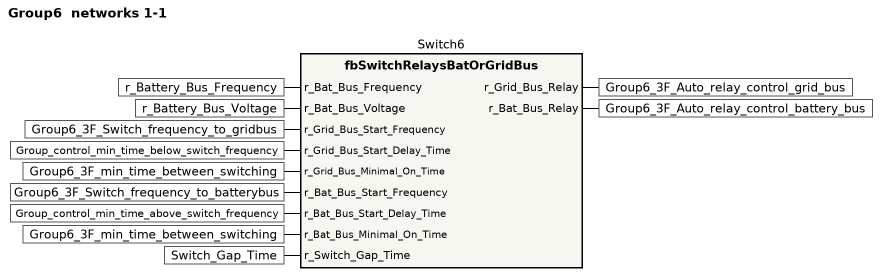
_FBD_ (* Function Block Diagram *)
NETWORK 1
	Switch6:fbSwitchRelaysBatOrGridBus(r_Bat_Bus_Frequency: r_Battery_Bus_Frequency, r_Bat_Bus_Voltage: r_Battery_Bus_Voltage, r_Grid_Bus_Start_Frequency: Group6_3F_Switch_frequency_to_gridbus, r_Grid_Bus_Start_Delay_Time: Group_control_min_time_below_switch_frequency, r_Grid_Bus_Minimal_On_Time: Group6_3F_min_time_between_switching, r_Bat_Bus_Start_Frequency: Group6_3F_Switch_frequency_to_batterybus, r_Bat_Bus_Start_Delay_Time: Group_control_min_time_above_switch_frequency, r_Bat_Bus_Minimal_On_Time: Group6_3F_min_time_between_switching, r_Switch_Gap_Time: Switch_Gap_Time, r_Bat_Bus_Relay => Group6_3F_Auto_relay_control_battery_bus) => Group6_3F_Auto_relay_control_grid_bus
_END_FBD_
(* the same logic as Structured Text *)
(* Network 1 *)
Switch6(r_Bat_Bus_Frequency := r_Battery_Bus_Frequency, r_Bat_Bus_Voltage := r_Battery_Bus_Voltage, r_Grid_Bus_Start_Frequency := Group6_3F_Switch_frequency_to_gridbus, r_Grid_Bus_Start_Delay_Time := Group_control_min_time_below_switch_frequency, r_Grid_Bus_Minimal_On_Time := Group6_3F_min_time_between_switching, r_Bat_Bus_Start_Frequency := Group6_3F_Switch_frequency_to_batterybus, r_Bat_Bus_Start_Delay_Time := Group_control_min_time_above_switch_frequency, r_Bat_Bus_Minimal_On_Time := Group6_3F_min_time_between_switching, r_Switch_Gap_Time := Switch_Gap_Time);
Group6_3F_Auto_relay_control_battery_bus := Switch6.r_Bat_Bus_Relay;
Group6_3F_Auto_relay_control_grid_bus := Switch6.r_Grid_Bus_Relay;
END_PROGRAM

(* POU 04. Frequency based Bus Select/Group7, FBD *)
PROGRAM Group7
VAR
	Switch7:fbSwitchRelaysBatOrGridBus;
END_VAR
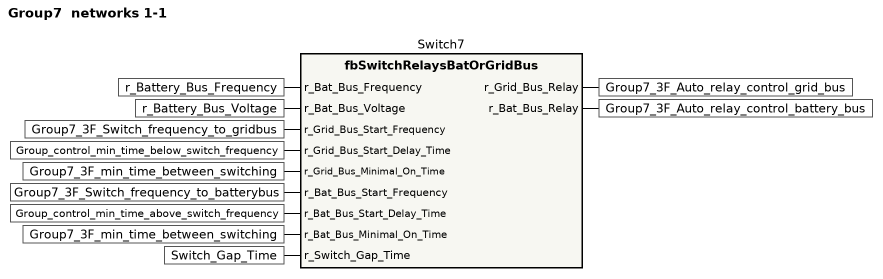
_FBD_ (* Function Block Diagram *)
NETWORK 1
	Switch7:fbSwitchRelaysBatOrGridBus(r_Bat_Bus_Frequency: r_Battery_Bus_Frequency, r_Bat_Bus_Voltage: r_Battery_Bus_Voltage, r_Grid_Bus_Start_Frequency: Group7_3F_Switch_frequency_to_gridbus, r_Grid_Bus_Start_Delay_Time: Group_control_min_time_below_switch_frequency, r_Grid_Bus_Minimal_On_Time: Group7_3F_min_time_between_switching, r_Bat_Bus_Start_Frequency: Group7_3F_Switch_frequency_to_batterybus, r_Bat_Bus_Start_Delay_Time: Group_control_min_time_above_switch_frequency, r_Bat_Bus_Minimal_On_Time: Group7_3F_min_time_between_switching, r_Switch_Gap_Time: Switch_Gap_Time, r_Bat_Bus_Relay => Group7_3F_Auto_relay_control_battery_bus) => Group7_3F_Auto_relay_control_grid_bus
_END_FBD_
(* the same logic as Structured Text *)
(* Network 1 *)
Switch7(r_Bat_Bus_Frequency := r_Battery_Bus_Frequency, r_Bat_Bus_Voltage := r_Battery_Bus_Voltage, r_Grid_Bus_Start_Frequency := Group7_3F_Switch_frequency_to_gridbus, r_Grid_Bus_Start_Delay_Time := Group_control_min_time_below_switch_frequency, r_Grid_Bus_Minimal_On_Time := Group7_3F_min_time_between_switching, r_Bat_Bus_Start_Frequency := Group7_3F_Switch_frequency_to_batterybus, r_Bat_Bus_Start_Delay_Time := Group_control_min_time_above_switch_frequency, r_Bat_Bus_Minimal_On_Time := Group7_3F_min_time_between_switching, r_Switch_Gap_Time := Switch_Gap_Time);
Group7_3F_Auto_relay_control_battery_bus := Switch7.r_Bat_Bus_Relay;
Group7_3F_Auto_relay_control_grid_bus := Switch7.r_Grid_Bus_Relay;
END_PROGRAM

(* POU 04. Frequency based Bus Select/Group8, FBD *)
PROGRAM Group8
VAR
	Switch8:fbSwitchRelaysBatOrGridBus;
END_VAR
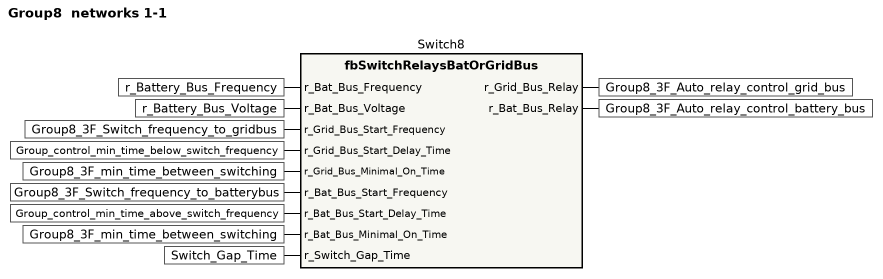
_FBD_ (* Function Block Diagram *)
NETWORK 1
	Switch8:fbSwitchRelaysBatOrGridBus(r_Bat_Bus_Frequency: r_Battery_Bus_Frequency, r_Bat_Bus_Voltage: r_Battery_Bus_Voltage, r_Grid_Bus_Start_Frequency: Group8_3F_Switch_frequency_to_gridbus, r_Grid_Bus_Start_Delay_Time: Group_control_min_time_below_switch_frequency, r_Grid_Bus_Minimal_On_Time: Group8_3F_min_time_between_switching, r_Bat_Bus_Start_Frequency: Group8_3F_Switch_frequency_to_batterybus, r_Bat_Bus_Start_Delay_Time: Group_control_min_time_above_switch_frequency, r_Bat_Bus_Minimal_On_Time: Group8_3F_min_time_between_switching, r_Switch_Gap_Time: Switch_Gap_Time, r_Bat_Bus_Relay => Group8_3F_Auto_relay_control_battery_bus) => Group8_3F_Auto_relay_control_grid_bus
_END_FBD_
(* the same logic as Structured Text *)
(* Network 1 *)
Switch8(r_Bat_Bus_Frequency := r_Battery_Bus_Frequency, r_Bat_Bus_Voltage := r_Battery_Bus_Voltage, r_Grid_Bus_Start_Frequency := Group8_3F_Switch_frequency_to_gridbus, r_Grid_Bus_Start_Delay_Time := Group_control_min_time_below_switch_frequency, r_Grid_Bus_Minimal_On_Time := Group8_3F_min_time_between_switching, r_Bat_Bus_Start_Frequency := Group8_3F_Switch_frequency_to_batterybus, r_Bat_Bus_Start_Delay_Time := Group_control_min_time_above_switch_frequency, r_Bat_Bus_Minimal_On_Time := Group8_3F_min_time_between_switching, r_Switch_Gap_Time := Switch_Gap_Time);
Group8_3F_Auto_relay_control_battery_bus := Switch8.r_Bat_Bus_Relay;
Group8_3F_Auto_relay_control_grid_bus := Switch8.r_Grid_Bus_Relay;
END_PROGRAM

(* POU 04. Frequency based Bus Select/Group9, FBD *)
PROGRAM Group9
VAR
	Switch9:fbSwitchRelaysBatOrGridBus;
END_VAR
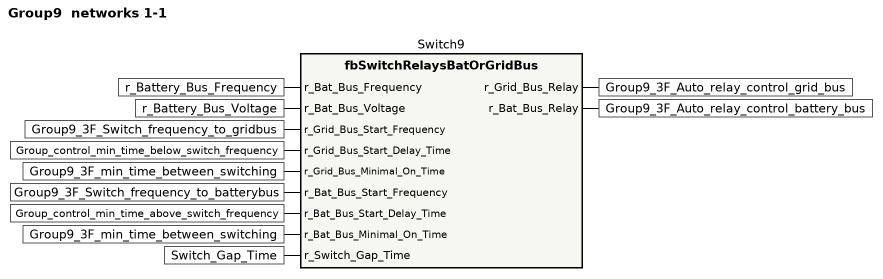
_FBD_ (* Function Block Diagram *)
NETWORK 1
	Switch9:fbSwitchRelaysBatOrGridBus(r_Bat_Bus_Frequency: r_Battery_Bus_Frequency, r_Bat_Bus_Voltage: r_Battery_Bus_Voltage, r_Grid_Bus_Start_Frequency: Group9_3F_Switch_frequency_to_gridbus, r_Grid_Bus_Start_Delay_Time: Group_control_min_time_below_switch_frequency, r_Grid_Bus_Minimal_On_Time: Group9_3F_min_time_between_switching, r_Bat_Bus_Start_Frequency: Group9_3F_Switch_frequency_to_batterybus, r_Bat_Bus_Start_Delay_Time: Group_control_min_time_above_switch_frequency, r_Bat_Bus_Minimal_On_Time: Group9_3F_min_time_between_switching, r_Switch_Gap_Time: Switch_Gap_Time, r_Bat_Bus_Relay => Group9_3F_Auto_relay_control_battery_bus) => Group9_3F_Auto_relay_control_grid_bus
_END_FBD_
(* the same logic as Structured Text *)
(* Network 1 *)
Switch9(r_Bat_Bus_Frequency := r_Battery_Bus_Frequency, r_Bat_Bus_Voltage := r_Battery_Bus_Voltage, r_Grid_Bus_Start_Frequency := Group9_3F_Switch_frequency_to_gridbus, r_Grid_Bus_Start_Delay_Time := Group_control_min_time_below_switch_frequency, r_Grid_Bus_Minimal_On_Time := Group9_3F_min_time_between_switching, r_Bat_Bus_Start_Frequency := Group9_3F_Switch_frequency_to_batterybus, r_Bat_Bus_Start_Delay_Time := Group_control_min_time_above_switch_frequency, r_Bat_Bus_Minimal_On_Time := Group9_3F_min_time_between_switching, r_Switch_Gap_Time := Switch_Gap_Time);
Group9_3F_Auto_relay_control_battery_bus := Switch9.r_Bat_Bus_Relay;
Group9_3F_Auto_relay_control_grid_bus := Switch9.r_Grid_Bus_Relay;
END_PROGRAM

(* POU 06. Mysql Write/Main_logger, ST *)
PROGRAM Main_logger
VAR


	xDoIt : BOOL;
	wState : WORD; (* Statemachine*)
	oMySql : MySql_Context; (* Used like Structure for keeping login and status information - Do not call it with in your program *)

	hasBufferedItems :  BOOL; (*Flag indicating the status of the buffer *)
	TONInst : TON; (* Sleep timer  *)

	(* Functionblock to contact MySql server *)
	oMySqlLogin : MySql_Login;

	xConnect : BOOL;
	diErrorLogin : DINT;
	sStatusLogin : STRING(500);
	xConnected : BOOL;

	(* Functionblock to process SQL statements who do not return result sets *)
	oMySqlExec1 : MySql_Execute;
	asSqlStatement1 : ARRAY [0..gcMySql_iSqlUpperBound] OF STRING(gcMySql_iSqlLength);
	xExec1 : BOOL;
	diErrorExec1 : DINT;
	sStatusExec1 : STRING(700);

	(*TODO clean this up these might be unnecassar delete if not used *)
	(* Functionblock to process SQL statements who return result sets *)
	oMySqlQuery1 : MySql_Query;
	asSqlQuery1 : ARRAY [0..gcMySql_iSqlUpperBound] OF STRING(gcMySql_iSqlLength);
	xQuery1 : BOOL;
	diErrorQuery1 : DINT;
	sStatusQuery1 : STRING(500);
	stQueryResult1 : MySql_ResultSet;

	(* Functionblock to disconnect MySql server *)
	oMySqlLogout : MySql_Logout;
	xDisconnect : BOOL;
	diErrorLogout : DINT;
	sStatusLogout : STRING(500);

	(* Helpers *)
	iHelp : INT;
	i : INT;
	END_: BOOL;
	strTempSQLStatement: STRING(raw_SQL_STR_LENGTH);


	(* debug variables *)
	iCountExecFailed: INT;
	xDolt: BOOL;

	stSystime: REAL;
END_VAR
(* Call function block "MySql_Login" every cycle to monitor connection status *)

oMySqlLogin(sHost:= gc_sHost,
			uiPort:= gc_uiPort,
			sUsername:= gc_sUser,
			sPassword:= gc_sPwd,
			sDatabase:=gc_sDB,
			oMySql:= oMySql,
			xStart:= xConnect,
			diError=> diErrorLogin,
			sStatus=> sStatusLogin,
			xConnected=> xConnected);

(*Get system time *)
(*
stSystime := Get_Time();
*)

CASE wState OF
0:

	xConnect := TRUE;
	wState := 10;

10:
	IF xConnected THEN

		xConnect := FALSE;
		IF TRUE  THEN  (*  Check that our power measurment model  is ready *)
			wState := 20; (* Proceede to execute SQL*)
		ELSE
			(* this is a different error state *)
			wState:= 45; (* wait and go to holding pattern for power measurement sensor to be ready*)
		END_IF
	ELSE
		wstate:=0;
	END_IF

20: (* prepare sql statement *)
	asSqlStatement1  := SQLStatement(    s_Table:= gc_sTable,
											);
	xExec1 := TRUE; (* Execute SQL-Insert-Statement *)
	wState :=25;

25:
	oMySqlExec1(asSqlCommand:=asSqlStatement1,
					oMySql:=oMySql,
					xStart:=xExec1,
					diError=> diErrorExec1,
					sStatus=>sStatusExec1);

	IF NOT  xExec1 THEN
		(* success *)
		xDisconnect := TRUE;
		wState := 50;  (*finished go and disconnect or start again *);

	ELSE

		(* Failed *)
		iCountExecFailed := iCountExecFailed +1; (* TODO count number of failures and fire an alarm *)
		wState:=50;

	END_IF


45: (* Wait here to debug convert problem *)
	(* buffer current value into memory *)
	(*
	IF gv_iBuffCounter < gc_MaxBufferSize THEN
		gv_Buffer[gv_iBuffCounter] := arCurrDataPoint; (* add data point to our buffer *)
		gv_iBuffCounter := gv_iBuffCounter + 1; (* incremenr buffer counter *)
		hasBufferedItems := TRUE; (*Flag indicating the status of the buffer *)
	END_IF
	*)
	wState := 46; (*move onto sleep*)

(*sleep X amount of time and continue*)


50: (* Disconnect from database *)
	oMySqlLogout(oMySql:= oMySql,
				 xStart:= xDisconnect,
				 diError=> diErrorLogout,
				 sStatus=> sStatusLogout);
	IF NOT xDisconnect THEN
		xDoIt := FALSE;
		wState := 60;(*move onto sleep*)



	END_IF

60:
	(*sleep X amount of time and continue*)
	TONInst( IN:= TRUE, PT := gc_LogInterval);

	IF TONInst.Q THEN
			wState := 0;
		(* do nothing just wait*)
	END_IF

END_CASE
END_PROGRAM

(* POU 06. Mysql Write/SQLStatement, ST *)
FUNCTION SQLStatement : ARRAY [0..gcMySql_iSqlUpperBound] OF STRING(gcMySql_iSqlLength)
VAR_INPUT

	s_Table 						: 	STRING;

END_VAR

VAR

	i	:	 INT;
	j	:	 INT;

	stNameArrayString	:	STRING;


END_VAR
SQLStatement[0] := 'INSERT INTO ';
SQLStatement[1] := s_Table;
SQLStatement[2] :=  '(datetime';

j:=3;
FOR i := 1 TO iNumberSystemVar DO

	SQLStatement[j] := CONCAT(',',(arSystemStateNames[i]));
	j:= j+1;

END_FOR

SQLStatement[j] := CONCAT(') VALUES (from_unixtime(',REAL_TO_STRING(arSystemState[0]));
j:=j+1;

SQLStatement[j] := ')';
j:=j+1;

FOR i := 1 TO iNumberSystemVar DO
	SQLStatement[j] :=  CONCAT(',',REAL_TO_STRING(arSystemState[i]));
	j:=j+1;
END_FOR

SQLStatement[j] :=  ');';
END_FUNCTION

(* POU Configuration/MODBUS_CONFIGURATION, ST *)
PROGRAM MODBUS_CONFIGURATION
VAR                                
END_VAR                            
(*
   <?xml version="1.0" encoding="UTF-16" standalone="yes"?>
<network xml_structure_version="1" xml_feature_version="1">
	<generator_settings minRTUTaskCycleTimeMs="100" minEthaskCycleTimeMs="5" ethSlaveMultiplier="0.1" rtuInterfaceMultiplier="0.1" taskGeneration="false"/>
	<master_interface type="serial" name="Configuration Root Node" com_port="2" baudrate="9600" databits="8" stopbits="1" parity="even" hwtype="RS485" flow_control="Xon/Xoff" asciimode="false" expanded="true">
		<mb_slave comment="" name="ModbusSlave" expanded="true" type="generic">
			<mb_connection type="serial" unitid="1" request_delay_ms="0" response_timeout_ms="1000"/>
			<generic_vars comment="" expanded="true">
				<generic_var data_type="REAL">
					<generic_params name="PhaseCurrenL2" comment="" expanded="false" mb_iotype="unused" mb_access="ro" var_byteorder="B3B4B1B2"/>
					<mb_address explicitAccess="false" FCRead="3" FCWrite="0" ReadMBAddress="20002" WriteMBAddress="0" ReadBitOffset="0" WriteBitOffset="0"/>
				</generic_var>
				<generic_var data_type="REAL">
					<generic_params name="VoltageV31" comment="" expanded="true" mb_iotype="unused" mb_access="ro" var_byteorder="B3B4B1B2"/>
					<mb_address explicitAccess="false" FCRead="3" FCWrite="0" ReadMBAddress="20012" WriteMBAddress="0" ReadBitOffset="0" WriteBitOffset="0"/>
				</generic_var>
				<generic_var data_type="REAL">
					<generic_params name="Pactive" comment="" expanded="true" mb_iotype="unused" mb_access="ro" var_byteorder="B3B4B1B2"/>
					<mb_address explicitAccess="false" FCRead="3" FCWrite="0" ReadMBAddress="20048" WriteMBAddress="0" ReadBitOffset="0" WriteBitOffset="0"/>
				</generic_var>
				<generic_var data_type="UINT">
					<generic_params name="ShortCircuitA" comment="" expanded="false" mb_iotype="unused" mb_access="ro" var_byteorder="B1B2B3B4"/>
					<mb_address explicitAccess="false" FCRead="3" FCWrite="0" ReadMBAddress="21002" WriteMBAddress="0" ReadBitOffset="0" WriteBitOffset="0"/>
				</generic_var>
				<generic_var data_type="UINT">
					<generic_params name="ShortCircuitB" comment="" expanded="true" mb_iotype="unused" mb_access="ro" var_byteorder="B1B2B3B4"/>
					<mb_address explicitAccess="false" FCRead="3" FCWrite="0" ReadMBAddress="21003" WriteMBAddress="0" ReadBitOffset="0" WriteBitOffset="0"/>
				</generic_var>
				<generic_var data_type="REAL">
					<generic_params name="Preactive" comment="" expanded="true" mb_iotype="unused" mb_access="ro" var_byteorder="B3B4B1B2"/>
					<mb_address explicitAccess="false" FCRead="3" FCWrite="0" ReadMBAddress="20050" WriteMBAddress="0" ReadBitOffset="0" WriteBitOffset="0"/>
				</generic_var>
				<generic_var data_type="UINT">
					<generic_params name="Phase1" comment="" expanded="false" mb_iotype="unused" mb_access="ro" var_byteorder="B1B2B3B4"/>
					<mb_address explicitAccess="false" FCRead="3" FCWrite="0" ReadMBAddress="21036" WriteMBAddress="0" ReadBitOffset="0" WriteBitOffset="0"/>
				</generic_var>
				<generic_var data_type="UINT">
					<generic_params name="Phase2" comment="" expanded="false" mb_iotype="unused" mb_access="ro" var_byteorder="B1B2B3B4"/>
					<mb_address explicitAccess="false" FCRead="3" FCWrite="0" ReadMBAddress="21037" WriteMBAddress="0" ReadBitOffset="0" WriteBitOffset="0"/>
				</generic_var>
				<generic_var data_type="UINT">
					<generic_params name="Phase3" comment="" expanded="false" mb_iotype="unused" mb_access="ro" var_byteorder="B1B2B3B4"/>
					<mb_address explicitAccess="false" FCRead="3" FCWrite="0" ReadMBAddress="21038" WriteMBAddress="0" ReadBitOffset="0" WriteBitOffset="0"/>
				</generic_var>
				<generic_var data_type="UINT">
					<generic_params name="StatusRemoteSwitching" comment="" expanded="false" mb_iotype="unused" mb_access="ro" var_byteorder="B1B2B3B4"/>
					<mb_address explicitAccess="false" FCRead="3" FCWrite="0" ReadMBAddress="23000" WriteMBAddress="0" ReadBitOffset="0" WriteBitOffset="0"/>
				</generic_var>
				<generic_var data_type="UINT">
					<generic_params name="SwitchLoadBreaker" comment="" expanded="true" mb_iotype="unused" mb_access="wo" var_byteorder="B1B2B3B4"/>
					<mb_address explicitAccess="false" FCRead="0" FCWrite="6" ReadMBAddress="0" WriteMBAddress="23100" ReadBitOffset="0" WriteBitOffset="0"/>
				</generic_var>
			</generic_vars>
		</mb_slave>
	</master_interface>
</network>
                              
*)                                 
;                                  
END_PROGRAM

(* POU 02. Batterybus Frequency to Analog Out/run_Frequency_Out, ST *)
PROGRAM run_Frequency_Out
VAR
END_VAR
CHP_Controller();
EV_Controller();
Mixer_Controller();
END_PROGRAM

(* POU 04. Frequency based Bus Select/run_group_switching, ST *)
PROGRAM run_group_switching
VAR
(*
	Group1 :fbSwitchRelaysBatOrGridBus; (* CHP Group has special rules *)
	Group2 :fbSwitchRelaysBatOrGridBus; (*  *)
	Group3 :fbSwitchRelaysBatOrGridBus; (*  *)
	Group4 :fbSwitchRelaysBatOrGridBus; (*  *)
	Group5 :fbSwitchRelaysBatOrGridBus; (*  *)
	Group6 :fbSwitchRelaysBatOrGridBus; (*  *)
	Group7 :fbSwitchRelaysBatOrGridBus; (*  *)
	Group8 :fbSwitchRelaysBatOrGridBus; (*  *)
	Group9 :fbSwitchRelaysBatOrGridBus; (*  *)
*)
END_VAR
(* frequency based switching is deactivated BY default AND can be activated via modbus *)

	Frequencybased_bus_selecting_state := REAL_TO_BOOL(arSystemState[261]) ;

	(* default switching gap time is 2000ms and can never be set lower than 500ms via Modbus *)
	Switch_Gap_Time								:= REAL_TO_INT(arSystemState[99]);
	IF Switch_Gap_Time < 500 THEN
		Switch_Gap_Time := 500;
	END_IF

(* group specific switch parameters (check modbus changes) *)
Group_control_Frequencybased_bus_selecting_state := arSystemState[246];
Group_control_min_time_above_switch_frequency := arSystemState[247];
Group_control_min_time_below_switch_frequency := arSystemState[248];
Group1_3F_Switch_frequency_to_batterybus := arSystemState[249];
Group1_3F_Switch_frequency_to_gridbus := arSystemState[250];
Group1_3F_min_time_between_switching := arSystemState[251];
Group2_3F_Switch_frequency_to_batterybus := arSystemState[252];
Group2_3F_Switch_frequency_to_gridbus := arSystemState[253];
Group2_3F_min_time_between_switching := arSystemState[254];
Group3_3F_Switch_frequency_to_batterybus := arSystemState[253];
Group3_3F_Switch_frequency_to_gridbus := arSystemState[254];
Group3_3F_min_time_between_switching := arSystemState[255];
Group4_3F_Switch_frequency_to_batterybus := arSystemState[256];
Group4_3F_Switch_frequency_to_gridbus := arSystemState[255];
Group4_3F_min_time_between_switching := arSystemState[256];
Group5_3F_Switch_frequency_to_batterybus := arSystemState[257];
Group5_3F_Switch_frequency_to_gridbus := arSystemState[258];
Group5_3F_min_time_between_switching := arSystemState[257];
Group6_3F_Switch_frequency_to_batterybus := arSystemState[258];
Group6_3F_Switch_frequency_to_gridbus := arSystemState[259];
Group6_3F_min_time_between_switching := arSystemState[260];
Group7_3F_Switch_frequency_to_batterybus := arSystemState[259];
Group7_3F_Switch_frequency_to_gridbus := arSystemState[260];
Group7_3F_min_time_between_switching := arSystemState[261];
Group8_3F_Switch_frequency_to_batterybus := arSystemState[262];
Group8_3F_Switch_frequency_to_gridbus := arSystemState[261];
Group8_3F_min_time_between_switching := arSystemState[262];
Group9_3F_Switch_frequency_to_batterybus := arSystemState[263];
Group9_3F_Switch_frequency_to_gridbus := arSystemState[264];
Group9_3F_min_time_between_switching := arSystemState[263];

IF Frequencybased_bus_selecting_state THEN
	Group1();
	Group2();
	Group3();
	Group4();
	Group5();
	Group6();
	Group7();
	Group8();
	Group9();
END_IF
END_PROGRAM

(* POU 03. Synchroniser Switch control/run_synchroniser_swtich, ST *)
PROGRAM run_synchroniser_swtich
VAR
END_VAR
SynchroniserSwitch();
END_PROGRAM

(* POU 05. System State Array/run_system_state_array, ST *)
PROGRAM run_system_state_array
VAR
END_VAR
variables_to_system_array();
END_PROGRAM

(* POU 03. Synchroniser Switch control/SynchronizerModbusStateHandler_PRG, ST *)
PROGRAM SynchronizerModbusStateHandler_PRG
VAR

END_VAR
(*___OLD___
IF r_modbus_Synchroniser_state < 1 THEN
		r_modbus_Synchroniser_Denied_Request := TRUE;
		r_modbus_Synchroniser_Close_Request := FALSE;
ELSE
	IF r_modbus_Synchroniser_state > 1.99 THEN
		r_modbus_Synchroniser_Denied_Request := FALSE;
		r_modbus_Synchroniser_Close_Request := TRUE;
	ELSE
		r_modbus_Synchroniser_Denied_Request := FALSE;
		r_modbus_Synchroniser_Close_Request := FALSE;
	END_IF
END_IF
*)
END_PROGRAM

(* POU 04. Frequency based Bus Select/Test, ST *)
PROGRAM Test
VAR

	Test :fbSwitchRelaysBatOrGridBus;
	a: REAL;
	frequencybased_bus_selecting_state: BOOL;
END_VAR
	frequencybased_bus_selecting_state : = arSystemState[999]; (* frequency based switching is deactivated by default and can be activated via modbus *)


Test(
	r_Off_Grid_Bus_Frequency:= r_Battery_Bus_Frequency ,
	r_Off_Grid_Bus_Voltage:= 250,
	r_On_Grid_Start_Frequency:= 49,
	r_On_Grid_Start_Delay_Time:= 2000,
	r_On_Grid_Minimal_On_Time:= 2000 ,
	r_Off_Grid_Start_Frequency:= 51,
	r_Off_Grid_Start_Delay_Time:= 2000,
	r_Switch_Gap_Time:= 2000,
	r_Off_Grid_Minimal_On_Time:= 2000);

(*
	Group1_Switch_frequency_to_batterybus						:  read from mobus;
	Group1_Switch_frequency_to_gridbus							:  REAL 	:= 48;
	Group1_min_time_above_switch frequency						:  INT 		: = 10000; (*ms*)
	Group1_min_time_below_switch frequency						:  INT 		: = 10000; (*ms*)
	Group1_min_time_between_switching							:  INT 		: = 10000; (*ms*)
*)
END_PROGRAM

(* POU 08. SD CARD logging/WriteCSVFile, ST *)
PROGRAM WriteCSVFile
(* 	This function block Writes the contents of the data structure to a CSV File

	Required Libraries:
		Standard.lib
		SysLibFile.lib
*)
VAR_INPUT
	sFILENAME 		:STRING(80); (* Filename to store data to (e.g. 'config.csv' 		*)
	typData			:ARRAY [1..iMaxParams] OF typCSV;
	bSeperator		:BYTE :=59;	(* Seperator semicolon:59=;*)
END_VAR
VAR_IN_OUT
	xStart 			:BOOL;	(* Set TRUE to write data, set False to stop.		 *)
END_VAR
VAR_OUTPUT
	sStatus			:STRING;
	iError 			:INT;	(* 00 : Normal Operation	*)
							(* 90 : Can't Open File 	*)
							(* 91 : Can't Close File 	*)
							(* 92 : Can't Write to File 	*)
END_VAR
VAR
	FileOpen		:BOOL := FALSE;
	handle			:DWORD;
	Mode			:STRING[20] := 'rw'; (* read/write *)
	DataString 		:STRING(80);
	i				:INT;
END_VAR
IF xStart THEN
	sStatus := 'Try to open file';
	IF NOT FileOpen THEN
		(* Open File *)
		handle := SysFileOpen(sFileName, Mode);
		IF handle > 0 THEN
			FileOpen := TRUE;
			sStatus := 'File Open OK.';
		ELSE
			iERROR := 90; (* Could not open file. *)
			sStatus := 'Could not open file.';
		END_IF
	END_IF
	
	IF FileOpen THEN
		FOR i := 1 TO iMaxParams DO
				DataString := TypData[i].sDescription;
				DataString := CONCAT(DataString,ASCIIBYTE_TO_STRING(bSeperator));
				DataString := CONCAT(DataString,(TypData[i].Parameter[1]));
	
				DataString := CONCAT(DataString,ASCIIBYTE_TO_STRING(13)); (* CR *)
				DataString := CONCAT(DataString,ASCIIBYTE_TO_STRING(10)); (* LF *)
				(* Write string to file *)
				IF SysFileWrite(handle, ADR(DataString), LEN(DataString)) = 0 THEN
					iERROR := 92; (* Could not write to file *)
					sStatus := 'Could not write file.';
				END_IF
		END_FOR
	END_IF
	
	IF FileOpen THEN
		(* Close file *)
		IF SysFileClose(handle) THEN
			FileOpen := FALSE;
			sStatus := 'File Saved.';
		ELSE
			iERROR := 91; (* Could not close file *)
			sStatus := 'Could not close file.';
		END_IF
		xStart := FALSE;
	END_IF
END_IF
END_PROGRAM

(* POU 06. Mysql Write/Create_Data_Point, ST *)
FUNCTION Create_Data_Point : DataPoint
VAR
		arCurrDataPoint   : DataPoint;
END_VAR
VAR_INPUT

	iSiteCode: INT;
	rTotalApparentPower				: REAL;						(* Total Apparent Power													II Scheinleistung gesamt *)
	rTotalPowerFactorPF				: REAL;						(* Total Power Factor PF 													II Leistungsfaktor_PF gesamt *)

	arFrequency						: ARRAY[1..3] OF REAL;		(* Frequency																II Frequenz *)
	arVoltage_L_N					: ARRAY[1..3] OF REAL;		(* Voltage L-N 																II Spannung Lx N *)
	arCurrent							: ARRAY[1..3] OF REAL;		(* Current 															   		II Strom *)

	(* TODO add the time stamp into buffered items*)

	DCV1 :REAL;
	DCV2 :REAL;

	DCPower1: REAL;
	DCPower2: REAL;

	DCCurr1 : REAL;
	DCCurr2 : REAL;


END_VAR
VAR
END_VAR
	arCurrDataPoint.iSiteCode := iSiteCode;
	arCurrDataPoint.rTotalApparentPower:=rTotalApparentPower;
	arCurrDataPoint.rTotalPowerFactorPF:=rTotalPowerFactorPF;

	arCurrDataPoint.arFrequency_1:=arFrequency[1];
	arCurrDataPoint.arVoltage_L_N_1:=arVoltage_L_N[1];
	arCurrDataPoint.arCurrent_1:=arCurrent[1];
	arCurrDataPoint.arPower_1:=arCurrDataPoint.arCurrent_1*arCurrDataPoint.arVoltage_L_N_1;

	arCurrDataPoint.arFrequency_2:=arFrequency[2];
	arCurrDataPoint.arVoltage_L_N_2:=arVoltage_L_N[2];
	arCurrDataPoint.arCurrent_2:=arCurrent[2];
	arCurrDataPoint.arPower_2:=arCurrDataPoint.arCurrent_2*arCurrDataPoint.arVoltage_L_N_2;


	arCurrDataPoint.arFrequency_3:=arFrequency[3];
	arCurrDataPoint.arVoltage_L_N_3:=arVoltage_L_N[3];
	arCurrDataPoint.arCurrent_3:=arCurrent[3];
	arCurrDataPoint.arPower_3:=arCurrDataPoint.arCurrent_3*arCurrDataPoint.arVoltage_L_N_3;

	arCurrDataPoint.timeStamp := Get_Time();

	arCurrDataPoint.DCV1 := DCV1;
	arCurrDataPoint.DCV2:=DCV2;
	arCurrDataPoint.DCPower1:=DCPower1;
	arCurrDataPoint.DCPower2:=DCPower2;
	arCurrDataPoint.DCCurr2:=DCCurr2;
	arCurrDataPoint.DCCurr2:=DCCurr2;


	Create_Data_Point := arCurrDataPoint;
END_FUNCTION

(* POU 06. Mysql Write/Get_Time, ST *)
FUNCTION Get_Time : REAL
VAR_INPUT

END_VAR
VAR



END_VAR
(* Haal de systeemtijd op *)
Get_Time := DT_TO_REAL(SysRtcGetTime(FALSE));
END_FUNCTION
